FUNCTION_BLOCK FB_Sorter
VAR_INPUT
END_VAR
VAR_OUTPUT
END_VAR
VAR
	on : BOOL;
	
	rTrigAtExit : Tc2_Standard.R_TRIG;
	exitTrigger : BOOL;
	atExitEdgeDetected : BOOL;
	
	Step_0_Standby : BOOL;
	Step_1 : BOOL;
	Step_2 : BOOL;
	Step_3 : BOOL;
	Step_4 : BOOL;
	Step_5 : BOOL;
	Step_6 : BOOL;
	Step_7 : BOOL;
	Step_10 : BOOL;
	Step_15 : BOOL;
	step_last : BOOL;
	
	dummy : BOOL;
	
	condition : BOOL;
	
	Opstart_puls_OS : BOOL;

	Initialiser_SQ: BOOL;
END_VAR
VAR_IN_OUT
	control_data : PlantAndCMs.Udt_PlantControl_Mode_1;
	
	control_data_vision : CM_Vision_UDT;
	control_data_Conveyor2 : CM_DO_UDT;
	
	control_data_sorter1 : CM_DO_UDT;
	control_data_sorter2 : CM_DO_UDT;
	control_data_sorter3 : CM_DO_UDT;
	
	control_data_atExit : CM_DIN_UDT;
	
	
END_VAR
VAR // added by the converter: edge detectors and wires of the graphical bodies
    _w1, _w2, _w3, _w4, _w5, _w6, _w7, _w8, _w9, _w10, _w11 : BOOL;
END_VAR

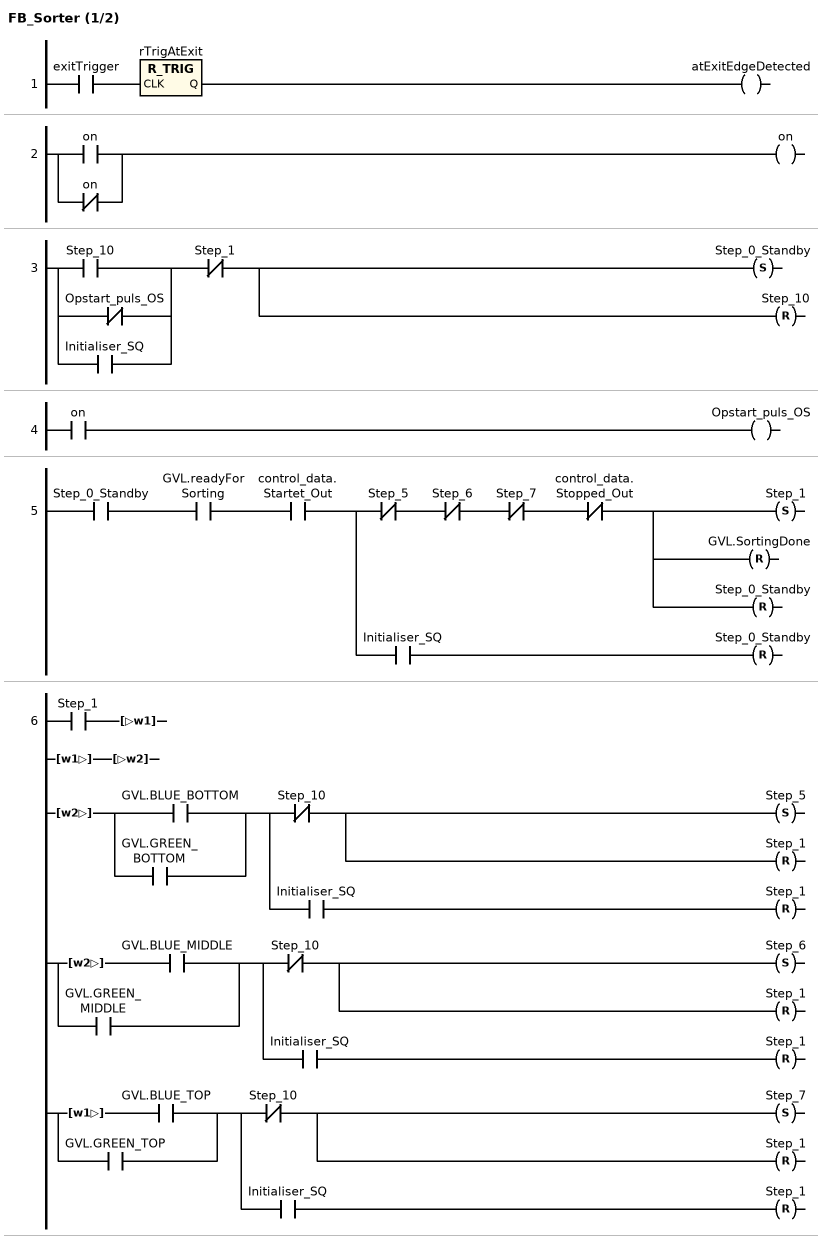
// NETWORK 1
rTrigAtExit(CLK := exitTrigger); // R_TRIG
atExitEdgeDetected := rTrigAtExit.Q;

// NETWORK 2
on := on OR NOT on;

// NETWORK 3
_w1 := (Step_10 OR NOT Opstart_puls_OS OR Initialiser_SQ) AND NOT Step_1;
Step_0_Standby S= _w1;
Step_10 R= _w1;

// NETWORK 4
Opstart_puls_OS := on;

// NETWORK 5
_w2 := Step_0_Standby AND GVL.readyForSorting AND control_data.Startet_Out;
_w3 := _w2 AND NOT Step_5 AND NOT Step_6 AND NOT Step_7 AND NOT control_data.Stopped_Out;
Step_1 S= _w3;
GVL.SortingDone R= _w3;
Step_0_Standby R= _w3;
Step_0_Standby R= _w2 AND Initialiser_SQ;

// NETWORK 6
_w4 := Step_1;
_w5 := _w4 AND (GVL.BLUE_BOTTOM OR GVL.GREEN_BOTTOM);
_w6 := _w5 AND NOT Step_10;
Step_5 S= _w6;
Step_1 R= _w6;
Step_1 R= _w5 AND Initialiser_SQ;
_w7 := _w4 AND GVL.BLUE_MIDDLE OR GVL.GREEN_MIDDLE;
_w8 := _w7 AND NOT Step_10;
Step_6 S= _w8;
Step_1 R= _w8;
Step_1 R= _w7 AND Initialiser_SQ;
_w9 := _w4 AND GVL.BLUE_TOP OR GVL.GREEN_TOP;
_w10 := _w9 AND NOT Step_10;
Step_7 S= _w10;
Step_1 R= _w10;
Step_1 R= _w9 AND Initialiser_SQ;

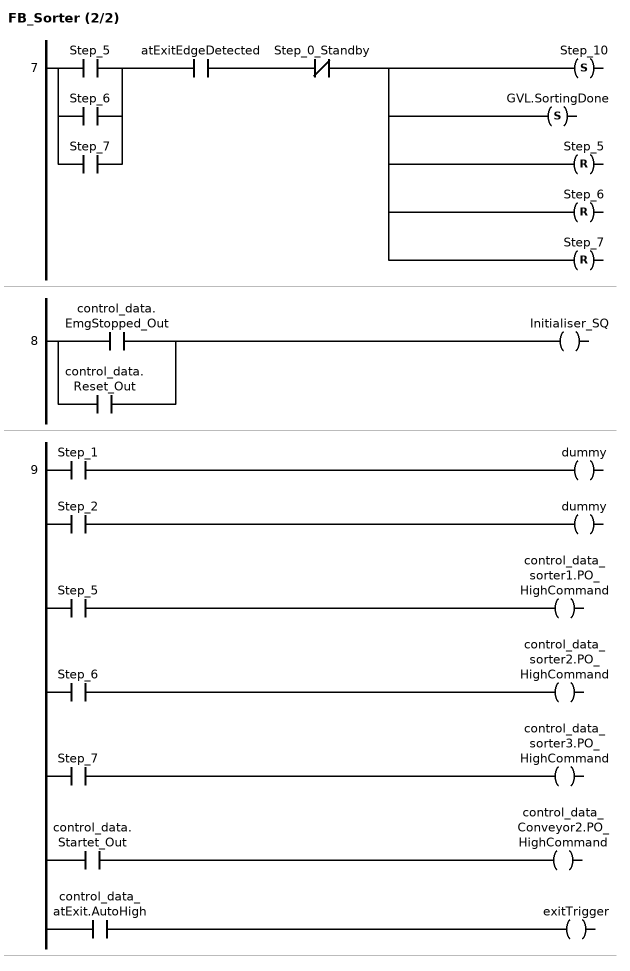
// NETWORK 7
_w11 := (Step_5 OR Step_6 OR Step_7) AND atExitEdgeDetected AND NOT Step_0_Standby;
Step_10 S= _w11;
GVL.SortingDone S= _w11;
Step_5 R= _w11;
Step_6 R= _w11;
Step_7 R= _w11;

// NETWORK 8
Initialiser_SQ := control_data.EmgStopped_Out OR control_data.Reset_Out;

// NETWORK 9
dummy := Step_1;
dummy := Step_2;
control_data_sorter1.PO_HighCommand := Step_5;
control_data_sorter2.PO_HighCommand := Step_6;
control_data_sorter3.PO_HighCommand := Step_7;
control_data_Conveyor2.PO_HighCommand := control_data.Startet_Out;
exitTrigger := control_data_atExit.AutoHigh;

END_FUNCTION_BLOCK

(* stored: Version 1.1.0.1, ProductVersion 3.1.4024.13
   POU FB_Sorter: Id {495ed67c-a59d-48ee-aabf-bc1a273d4fac}, SpecialFunc None *)
